(* IEC 61131-3 sources: test/Class/Sfc_StepInvoker, 1 file *)

(* ---- Sfc_StepInvoker.st ---- *)
#define MAX_STEP_CNT 1000
#define MAX_ACTIVE_STEP_CNT 100

(*!
<Class
	Name               = "Sfc_StepInvoker"
	Revision           = "1.0"
	RealtimeTask       = "false"
	CyclicTask         = "false"
	BackgroundTask     = "false"
	Sigmatek           = "true"
	OSInterface        = "false"
	HighPriority       = "false"
	Automatic          = "false"
	UpdateMode         = "Prescan"
	SharedCommandTable = "true"
	Objectsize         = "(284,120)"
	Comment            = "Handles step execution">
	<Channels>
		<Server Name="LogonItf" Visualized="false" Initialize="false" WriteProtected="false" Retentive="false" Comment="Interface to the stepinvoker class&#13;&#10;&#13;&#10;Steps use this server to register themselves"/>
	</Channels>
</Class>
*)
Sfc_StepInvoker : CLASS
	TYPE
	  StepPtr : ^Sfc_Step_Base;
	  ActiveStepArray : ARRAY [0..MAX_ACTIVE_STEP_CNT] OF StepPtr;
	  StepArray : ARRAY [0..MAX_STEP_CNT] OF StepPtr;
	END_TYPE
  //Servers:
	LogonItf 	: SvrChCmd_pVoid;
  //Clients:
  //Variables:
		m_Steps 	: StepArray;
		m_StepCnt 	: DINT;
		m_ActiveSteps 	: ActiveStepArray;
		m_ActiveStepCnt 	: DINT;
  //Functions:

	FUNCTION Sfc_StepInvoker
		VAR_OUTPUT
			ret_code 	: ConfStates;
		END_VAR;

	FUNCTION GLOBAL Work;

	FUNCTION VIRTUAL GLOBAL LogonItf::Write
		VAR_INPUT
			input (EAX) 	: pVoid;
		END_VAR
		VAR_OUTPUT
			result (EAX) 	: pVoid;
		END_VAR;
  //Tables:
	FUNCTION @STD
		VAR_OUTPUT
			ret_code	: CONFSTATES;
		END_VAR;
	FUNCTION GLOBAL TAB @CT_;
END_CLASS;

#pragma usingLtd Sfc_Step_Base

FUNCTION Sfc_StepInvoker::Sfc_StepInvoker
	VAR_OUTPUT
		ret_code 	: ConfStates;
	END_VAR
  VAR
	  index : DINT;
  END_VAR

  m_StepCnt := 0;
  m_ActiveStepCnt := 0;

  for index := 0 to MAX_STEP_CNT - 1 by 1 do

    m_Steps[index] := NIL;

  end_for;

	ret_code := C_OK;

END_FUNCTION

FUNCTION VIRTUAL GLOBAL Sfc_StepInvoker::LogonItf::Write
	VAR_INPUT
		input (EAX) 	: pVoid;
	END_VAR
	VAR_OUTPUT
		result (EAX) 	: pVoid;
	END_VAR

	if m_StepCnt < (MAX_STEP_CNT-1) then

    m_Steps[m_StepCnt] := input$StepPtr;

    m_StepCnt += 1;

    result := input;

  else

    result := NIL;

  end_if;

END_FUNCTION

FUNCTION GLOBAL Sfc_StepInvoker::Work
  VAR
	  index : DINT;
    pStep : ^StepPtr;
  END_VAR

  m_ActiveStepCnt := 0;

  //////////////////////////////////////////////////////////////
  // Determine list of active steps

  // Initialize Pointer
  pStep := #m_Steps$StepPtr;

  for index := 0 to m_StepCnt - 1 by 1 do

    if pStep^^.X then

      m_ActiveSteps[m_ActiveStepCnt] := pStep^;

      m_ActiveStepCnt += 1;

    end_if;

    // Next Element
    pStep += sizeof(StepPtr);

  end_for;

  // Determine list of active steps
  //////////////////////////////////////////////////////////////

  //////////////////////////////////////////////////////////////
  // Execute work routine of active steps

  // Initialize Pointer
  pStep := #m_ActiveSteps$StepPtr;

  for index := 0 to m_ActiveStepCnt - 1 by 1 do

    pStep^^.Work();

    // Next Element
    pStep += sizeof(StepPtr);

  end_for;

  // Execute work routine of active steps
  //////////////////////////////////////////////////////////////

END_FUNCTION
